{attribute 'linkalways'} 
{attribute 'no_explicit_call' := 'This FB is a CLASS and must be accessed using methods or properties'}
{attribute 'enable_dynamic_creation'}
FUNCTION_BLOCK Scene
VAR
	animations : Queue;
	elements : Queue;
END_VAR

METHOD PUBLIC AddAnimation
VAR_INPUT
	GraphicalElement : I_GraphicalElement;
END_VAR
elements.Enqueue(GraphicalElement);
END_METHOD

METHOD PUBLIC AddElement
VAR_INPUT
	GraphicalElement : I_GraphicalElement;
END_VAR
elements.Enqueue(GraphicalElement);
END_METHOD

METHOD Clear
VAR_INPUT
END_VAR
elements.Clear();
END_METHOD

METHOD PUBLIC RenderTo
VAR_INPUT
	Destination : I_WritableDisplayBuffer;
END_VAR
VAR
	enumerator : I_ForwardEnumerator;
	element : I_GraphicalElement;
END_VAR
enumerator := elements.GetEnumerator();

WHILE enumerator.MoveNext() DO
	IF enumerator.TryGet(element) THEN
		element.RenderTo(Destination);
	END_IF
END_WHILE

enumerator.Dispose();
END_METHOD

METHOD PUBLIC TryRemoveElement : BOOL
VAR_INPUT
	GraphicalElement : I_GraphicalElement;
END_VAR
TryRemoveElement := elements.TryRemoveItem(GraphicalElement);
END_METHOD

METHOD PUBLIC Update
VAR_INPUT
	DeltaTimeInMs : UDINT;
END_VAR
VAR
	enumerator : I_ForwardEnumerator;
	element : I_GraphicalElement;
END_VAR
enumerator := elements.GetEnumerator();

WHILE enumerator.MoveNext() DO
	IF enumerator.TryGet(element) THEN
		element.Update(DeltaTimeInMs);
	END_IF
END_WHILE

enumerator.Dispose();
END_METHOD

END_FUNCTION_BLOCK

(* stored: Version 1.1.0.1, ProductVersion 3.1.4024.15
   POU Scene: Id {47179599-057e-40d4-8e43-57f30a2a9f4f}, SpecialFunc None
   Method AddAnimation: Id {c36236e6-f121-476c-9666-787c5f51975e}
   Method AddElement: Id {bfc35db7-ee79-4972-b28b-1ceb29d3437f}
   Method Clear: Id {99019aaf-97e0-4529-bccf-c35ea48986c2}
   Method RenderTo: Id {e7e2245b-7946-4791-ae16-16da2564931f}
   Method TryRemoveElement: Id {3a32d136-e86d-4332-8582-d02683c0e6c0}
   Method Update: Id {6848dc00-eb64-426f-abf8-9d8525aefce0} *)
